PROGRAM MAIN
VAR CONSTANT
	sLogger		: STRING := 'MAIN';
END_VAR
VAR
	nCounter	: UINT;
	fbCountTime	: TON := (PT:=T#1S);
END_VAR

IF _TaskInfo[GETCURTASKINDEXEX()].FirstCycle THEN
	F_LogL(E_LogLevel.eInfo, sLogger, 'SPS Task gestartet.');
END_IF

fbCountTime(IN:=NOT fbCountTime.Q);
IF fbCountTime.Q THEN
	nCounter := nCounter + 1;
	F_LogLA1C(
		E_LogLevel.eDebug, 
		sLogger, 
		'Zähler geändert, neuer Wert {0}', 
		nCounter, 
		F_LogContext().AddInt('MachineNo', 42)
	);
END_IF

PRG_TaskLog.Call();

END_PROGRAM

(* stored: Version 1.1.0.1, ProductVersion 3.1.4024.0
   POU MAIN: Id {14a21c79-1aea-4be4-b206-ffa0d92e1c5a}, SpecialFunc None *)
